screen "Screen_1" 1366x768
   GraphicView "Graphic view_5" at 263,400 size 357x69; Picture "Graphic_8"
   GraphicView "Graphic view_1" at 245,95 size 177x231; Picture "Graphic_1"
   Button "Button_1" at 5,4 size 130x36; TextOff 'Exit SCADA'
      on Press: StopRuntime(0)
   GraphicView "Graphic view_2" at 401,14 size 67x78; Picture "Graphic_2"
   GraphicView "Graphic view_3" at 209,14 size 67x78; Picture "Graphic_2"
   GraphicView "Graphic view_12" at 358,60 size 46x48; Picture "Graphic_7"
   GraphicView "Graphic view_13" at 274,60 size 48x48; Picture "Graphic_5"
   GraphicView "Graphic view_14" at 462,57 size 103x30; Picture "Graphic_4"
   GraphicView "Graphic view_15" at 110,58 size 103x30; Picture "Graphic_4"
   TextField "Text field_1" at 167,13 size 46x23; Text 'V101'
   TextField "Text field_2" at 358,14 size 46x23; Text 'V102'
   Rectangle "Rectangle_1" at 227,19 size 31x16
      Visibility <- "V101_On"
   Rectangle "Rectangle_3" at 419,19 size 31x16
      Visibility <- "V102_On"
   Button "Button_2" at 598,8 size 168x64; TextOff 'Start'
      on Release: ResetBit("Start_PB")
      on Press: SetBit("Start_PB")
   Button "Button_7" at 600,81 size 168x64; TextOff 'Automatic'
      on Release: ResetBit("Auto_Mode")
      on Press: SetBit("Auto_Mode")
   Button "Button_4" at 600,152 size 168x64; TextOff 'Recipe 1'
      on Release: ResetBit("Recipe_1")
      on Press: SetBit("Recipe_1")
   GraphicView "Graphic view_4" at 416,296 size 65x72; Picture "Graphic_2"
   GraphicView "Graphic view_6" at 109,291 size 67x78; Picture "Graphic_2"
   GraphicView "Graphic view_7" at 306,319 size 52x43; Picture "Graphic_3"
   GraphicView "Graphic view_8" at 355,333 size 66x35; Picture "Graphic_4"
   GraphicView "Graphic view_9" at 475,342 size 37x36; Picture "Graphic_5"
   GraphicView "Graphic view_10" at 172,332 size 140x38; Picture "Graphic_6"
   GraphicView "Graphic view_11" at 62,336 size 50x46; Picture "Graphic_7"
   TextField "Text field_3" at 481,307 size 46x23; Text 'V103'
   TextField "Text field_4" at 63,291 size 46x23; Text 'V104'
   GraphicView "Graphic view_16" at 378,122 size 90x167; Picture "Graphic_9"
   TextField "Text field_5" at 429,108 size 51x23; Text 'Mixer'
   GraphicView "Graphic view_17" at 249,238 size 42x64; Picture "Graphic_11"
   TextField "Text field_6" at 188,226 size 61x23; Text 'Heater'
   GraphicView "Graphic view_18" at 481,382 size 50x52; Picture "Graphic_12"
   GraphicView "Graphic view_19" at 418,383 size 50x52; Picture "Graphic_12"
   GraphicView "Graphic view_20" at 355,384 size 50x52; Picture "Graphic_12"
   Rectangle "Rectangle_5" at 126,296 size 31x16
      Visibility <- "V104_On"
   Rectangle "Rectangle_7" at 433,300 size 31x16
      Visibility <- "V103_On"
   Rectangle "Rectangle_10" at 455,173 size 31x16
      Visibility <- "Mixer_On"
   Rectangle "Rectangle_9" at 273,220 size 31x16
      Visibility <- "Heater_On"
   Button "Button_3" at 600,152 size 168x64; TextOff 'Recipe 1'
      on Release: ResetBit("Recipe_1")
      on Press: SetBit("Recipe_1")
   Button "Button_5" at 601,224 size 168x64; TextOff 'Recipe 2'
      on Release: ResetBit("Recipe_2")
      on Press: SetBit("Recipe_2")
   Button "Button_6" at 601,296 size 168x64; TextOff 'Recipe 3'
      on Release: ResetBit("Recipe_3")
      on Press: SetBit("Recipe_3")
   IOField "I/O field_1" at 263,409 size 86x25; FormatPattern s99999
      ProcessValue <- "Bottle_Count"
   TextField "Text field_7" at 150,408 size 108x23; Text 'Bottle Count'
   Rectangle "Rectangle_2" at 301,443 size 31x16
      Visibility <- "Conveyor_On"
   Rectangle "Rectangle_4" at 356,443 size 31x16
      Visibility <- "Conveyor_On"
   Rectangle "Rectangle_6" at 414,443 size 31x16
      Visibility <- "Conveyor_On"
   Rectangle "Rectangle_8" at 470,443 size 31x16
      Visibility <- "Conveyor_On"
   Rectangle "Rectangle_11" at 528,443 size 31x16
      Visibility <- "Conveyor_On"
   IOField "I/O field_2" at 192,248 size 58x25; FormatPattern 99.99
      ProcessValue <- "Temperature_Measurement_In_PV"
   Button "Button_8" at 13,199 size 168x64; TextOff 'Reset'
      on Release: ResetBit("Reset_PB")
      on Press: SetBit("Reset_PB")
   Button "Button_9" at 13,130 size 168x64; TextOff 'Stop'
      on Release: ResetBit("Stop_PB")
      on Press: SetBit("Stop_PB")
   Button "Button_10" at 618,375 size 83x68; TextOff 'Bottle'
      on Release: ResetBit("Bottle_Sim_output")
      on Press: SetBit("Bottle_Sim_output")
   TextField "Text field_8" at 864,262 size 125x22; Text 'Recipe Selected'
   TextField "Text field_9" at 802,354 size 119x23; Text 'Product A (L):'
   TextField "Text field_10" at 802,286 size 128x23; Text 'Bottle Size (L):'
   TextField "Text field_11" at 802,319 size 117x23; Text 'No of Bottles:'
   TextField "Text field_12" at 802,388 size 118x23; Text 'Product B (L):'
   TextField "Text field_13" at 802,423 size 121x23; Text 'Mix Temp (C):'
   TextField "Text field_14" at 801,460 size 130x23; Text 'Mix Time (mS):'
   IOField "I/O field_4" at 507,156 size 67x25; FormatPattern s9999999999
      ProcessValue <- "Mixing_Timer_ET"
   TextField "Text field_15" at 512,131 size 53x23; Text 'Timer'
   IOField "I/O field_3" at 172,437 size 86x25; FormatPattern 99999
      ProcessValue <- "Conveyor_Speed_value"
   TextField "Text field_16" at 28,437 size 136x23; Text 'Conveyor Speed'
   IOField "I/O field_5" at 938,286 size 56x26; FormatPattern s999
      ProcessValue <- "Recipe Selection_DB_Bottle_Size"
   IOField "I/O field_6" at 938,322 size 55x26; FormatPattern s99999
      ProcessValue <- "Recipe Selection_DB_Bottle_Number"
   IOField "I/O field_7" at 937,354 size 55x26; FormatPattern s99999
      ProcessValue <- "Recipe Selection_DB_Product_A"
   IOField "I/O field_8" at 936,386 size 56x26; FormatPattern s99999
      ProcessValue <- "Recipe Selection_DB_Product_B"
   IOField "I/O field_9" at 936,423 size 56x26; FormatPattern s99999
      ProcessValue <- "Recipe Selection_DB_Mix_Temp"
   IOField "I/O field_10" at 936,460 size 76x26; FormatPattern s9999999999
      ProcessValue <- "Recipe Selection_DB_Mixing_Time"
   Circle "Circle_14" at 710,382 size 53x53
      Appearance <- "Bottle_Pos_OK"
   Rectangle "Rectangle_13" at 28,502 size 147x61
      Appearance <- "Step_1"
   Rectangle "Rectangle_15" at 763,502 size 147x61
      Appearance <- "Step_6"
   Rectangle "Rectangle_17" at 910,502 size 147x61
      Appearance <- "Step_8"
   Rectangle "Rectangle_18" at 175,502 size 147x61
      Appearance <- "Step_2"
   Rectangle "Rectangle_19" at 322,502 size 147x61
      Appearance <- "Step_3"
   Rectangle "Rectangle_20" at 469,502 size 147x61
      Appearance <- "Step_4"
   Rectangle "Rectangle_21" at 616,502 size 147x61
      Appearance <- "Step_5"
   Rectangle "Rectangle_22" at 1057,502 size 147x61
      Appearance <- "End_cycle"
   TextField "Text field_17" at 1064,513 size 135x40; Text 'End Of Cycle (Batch Complete)'
   TextField "Text field_18" at 66,512 size 66x40; Text 'Process Starting'
   TextField "Text field_19" at 210,514 size 77x40; Text 'Product A Filling'
   TextField "Text field_20" at 357,513 size 77x40; Text 'Product B Filling'
   TextField "Text field_21" at 500,512 size 91x40; Text 'Mixer and Heating ON'
   TextField "Text field_22" at 500,512 size 91x40; Text 'Mixer and Heating ON'
   TextField "Text field_23" at 656,512 size 69x40; Text 'Cooking Process'
   TextField "Text field_24" at 792,503 size 99x58; Text 'Conditioning Cycle Starting'
   TextField "Text field_26" at 957,513 size 52x40; Text 'Bottle Filling'
   TextField "Text field_28" at 1104,16 size 75x23; Text 'Recipe 1'
   TextField "Text field_29" at 1241,17 size 75x23; Text 'Recipe 2'
   TextField "Text field_30" at 1237,262 size 75x23; Text 'Recipe 3'
   TextField "Text field_31" at 805,111 size 267x23; Text 'Product A / Tolerance (+/-) (L):'
   TextField "Text field_32" at 805,43 size 128x23; Text 'Bottle Size (L):'
   TextField "Text field_33" at 805,76 size 117x23; Text 'No of Bottles:'
   TextField "Text field_34" at 805,145 size 266x23; Text 'Product B / Tolerance (+/-) (L):'
   TextField "Text field_35" at 805,180 size 269x23; Text 'Mix Temp / Tolerance (+/-) (C):'
   IOField "I/O field_11" at 1112,43 size 53x27; FormatPattern s99999
      ProcessValue <- "Bottle_Size_Rec1"
   IOField "I/O field_12" at 1247,294 size 53x27; FormatPattern s99999
      ProcessValue <- "Bottle_Size_Rec3"
   IOField "I/O field_13" at 1250,49 size 53x27; FormatPattern s99999
      ProcessValue <- "Bottle_Size_Rec2"
   IOField "I/O field_14" at 1112,70 size 53x27; FormatPattern s99999
      ProcessValue <- "Bottle_Batch_Size_Rec1"
   IOField "I/O field_15" at 1250,72 size 53x27; FormatPattern s99999
      ProcessValue <- "Bottle_Batch_Size_Rec2"
   IOField "I/O field_16" at 1247,323 size 53x27; FormatPattern s99999
      ProcessValue <- "Bottle_Batch_Size_Rec3"
   IOField "I/O field_17" at 1084,113 size 52x27; FormatPattern s99999
      ProcessValue <- "ProdA_SP_Rec1"
   IOField "I/O field_18" at 1137,113 size 52x27; FormatPattern s99999
      ProcessValue <- "ProdA_Tol_Rec1"
   IOField "I/O field_19" at 1223,113 size 52x27; FormatPattern s99999
      ProcessValue <- "ProdA_SP_Rec2"
   IOField "I/O field_20" at 1276,113 size 52x27; FormatPattern s99999
      ProcessValue <- "ProdA_Tol_Rec2"
   IOField "I/O field_21" at 1222,358 size 52x27; FormatPattern s99999
      ProcessValue <- "ProdA_SP_Rec3"
   IOField "I/O field_22" at 1275,358 size 52x27; FormatPattern s99999
      ProcessValue <- "ProdA_Tol_Rec3"
   IOField "I/O field_23" at 1084,141 size 52x27; FormatPattern s99999
      ProcessValue <- "ProdB_SP_Rec1"
   IOField "I/O field_24" at 1137,141 size 52x27; FormatPattern s99999
      ProcessValue <- "ProdB_Tol_Rec1"
   IOField "I/O field_25" at 1223,140 size 52x27; FormatPattern s99999
      ProcessValue <- "ProdB_SP_Rec2"
   IOField "I/O field_26" at 1276,140 size 52x27; FormatPattern s99999
      ProcessValue <- "ProdB_Tol_Rec2"
   IOField "I/O field_27" at 1222,384 size 52x27; FormatPattern s99999
      ProcessValue <- "ProdB_SP_Rec3"
   IOField "I/O field_28" at 1275,384 size 52x27; FormatPattern s99999
      ProcessValue <- "ProdB_Tol_Rec3"
   IOField "I/O field_29" at 1084,180 size 52x27; FormatPattern s99999
      ProcessValue <- "Mix_Temp_SP_Rec1"
   IOField "I/O field_30" at 1137,180 size 52x27; FormatPattern s99999
      ProcessValue <- "Mix_Temp_Tol_Rec1"
   IOField "I/O field_31" at 1086,216 size 104x27; FormatPattern 99999
      ProcessValue <- "Mix_Time_Rec1"
   IOField "I/O field_32" at 1223,176 size 52x27; FormatPattern s99999
      ProcessValue <- "Mix_Temp_SP_Rec2"
   IOField "I/O field_33" at 1276,176 size 52x27; FormatPattern s99999
      ProcessValue <- "Mix_Temp_Tol_Rec2"
   IOField "I/O field_34" at 1222,421 size 52x27; FormatPattern s99999
      ProcessValue <- "Mix_Temp_SP_Rec3"
   IOField "I/O field_35" at 1275,421 size 52x27; FormatPattern s99999
      ProcessValue <- "Mix_Temp_Tol_Rec3"
   IOField "I/O field_36" at 1223,462 size 102x27; FormatPattern 99999
      ProcessValue <- "Mix_Time_Rec3"
   IOField "I/O field_37" at 1224,216 size 103x27; FormatPattern 99999
      ProcessValue <- "Mix_Time_Rec2"
   TextField "Text field_36" at 805,220 size 130x23; Text 'Mix Time (mS):'
   TextField "Text field_37" at 1084,295 size 128x23; Text 'Bottle Size (L):'
   TextField "Text field_38" at 1085,323 size 117x23; Text 'No of Bottles:'
   TextField "Text field_39" at 1085,359 size 119x23; Text 'Product A (L):'
   TextField "Text field_40" at 1086,385 size 118x23; Text 'Product B (L):'
   TextField "Text field_41" at 1087,422 size 121x23; Text 'Mix Temp (C):'
   TextField "Text field_42" at 1087,462 size 121x23; Text 'Mix Temp (C):'
   Bar "Bar_2" at 318,124 size 69x174; MinimumValue 0; MaximumValue 1000
      ProcessValue <- "Ultrasonic_Lvl_In_DB_PV"
   Rectangle "Rectangle_14" at 29,592 size 147x61
      Appearance <- "ProdA_Level_Error"
   Rectangle "Rectangle_16" at 176,592 size 147x61
      Appearance <- "ProdB_Level_Error"
   Rectangle "Rectangle_25" at 323,592 size 147x61
      Appearance <- "Heater_liquid_error"
   TextField "Text field_25" at 57,611 size 97x22; Text 'Prod A Error'
   TextField "Text field_27" at 204,611 size 97x22; Text 'Prod B Error'
   TextField "Text field_43" at 349,603 size 95x40; Text 'Mixing Tank Level Error'
   Rectangle "Rectangle_26" at 470,592 size 147x61
      Appearance <- "Conveyor_error"
   TextField "Text field_44" at 506,602 size 80x40; Text 'Conveyor Error'
   Rectangle "Rectangle_27" at 617,592 size 147x61
      Appearance <- "Overflow_Error"
   TextField "Text field_45" at 643,603 size 103x40; Text 'Tank Overfill Error'
   Rectangle "Rectangle_28" at 763,592 size 147x61
      Appearance <- "EMS_Triggered"
   TextField "Text field_46" at 775,610 size 126x22; Text 'Emergengy Stop'
*)